(* Logix 5000 project; controller Nut_Filling_Station Emulate 5570 rev 33.11; software revision 33.03 *)

TASK MainTask (continuous, watchdog 500 ms) : MainProgram

MODULES
   Local : Emulate 5570 (ICP 3, rev 33.11)
END_MODULES

VAR_GLOBAL   (* controller tags *)
   Conveyor_Run : BOOL;   // Conveyor motor command
   Entry_PE : BOOL;   // Box at label-reading position
   Exit_PE : BOOL;   // Box at exit
   Green_Label : BOOL;   // Green label detected
   Peanut_Box_Count : COUNTER := (PRE := 1000);   // Counts completed peanut boxes
   Peanut_Filled_Up : BOOL;   // Peanut station reports target weight reached
   Peanut_Open : BOOL;   // Peanut hopper valve command
   Peanut_PE : BOOL;   // Box underneath peanut hopper
   Peanut_Total_kg : REAL;   // Total peanut kilograms packed
   Red_Label : BOOL;   // Red label detected
   Reset_Counts_PB : BOOL;   // Clears production counts
   Reset_PB : BOOL;   // Reset sequence
   Run_Enable : BOOL;   // Automatic operation enabled
   Start_PB : BOOL;   // Start pushbutton
   Step : DINT;   // Current sequence step
   Step_Scan : DINT;   // Step captured at start of this scan
   Stop_OK : BOOL;   // 1 when Stop is released
   Walnut_Box_Count : COUNTER := (PRE := 1000);   // Counts completed walnut boxes
   Walnut_Filled_Up : BOOL;   // Walnut station reports target weight reached
   Walnut_Open : BOOL;   // Walnut hopper valve command
   Walnut_PE : BOOL;   // Box underneath walnut hopper
   Walnut_Total_kg : REAL;   // Total walnut kilograms packed
END_VAR

PROGRAM MainProgram   (* main routine MainRoutine *)

ROUTINE MainRoutine   (* ladder *)
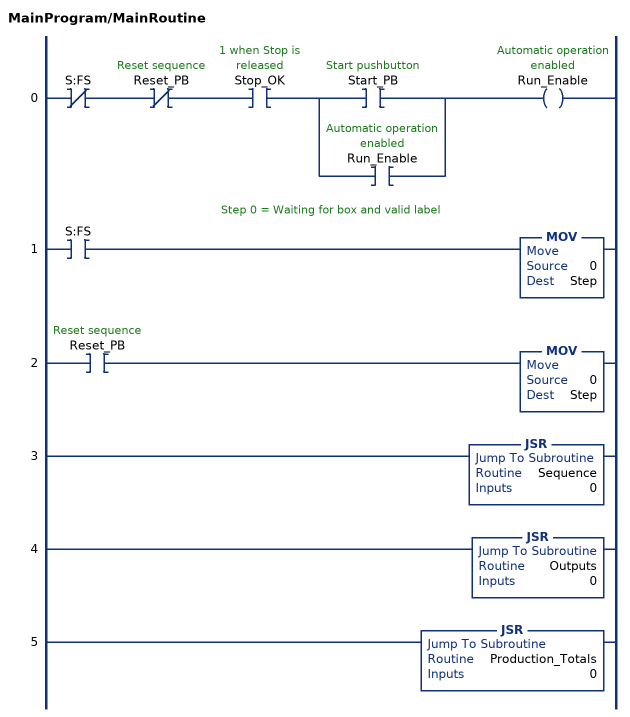
   0: XIO(S:FS)XIO(Reset_PB)XIC(Stop_OK)[XIC(Start_PB) ,XIC(Run_Enable) ]OTE(Run_Enable);
   // Step 0 = Waiting for box and valid label
   1: XIC(S:FS)MOV(0,Step);
   2: XIC(Reset_PB)MOV(0,Step);
   3: JSR(Sequence,0);
   4: JSR(Outputs,0);
   5: JSR(Production_Totals,0);
END_ROUTINE

ROUTINE Outputs   (* ladder *)
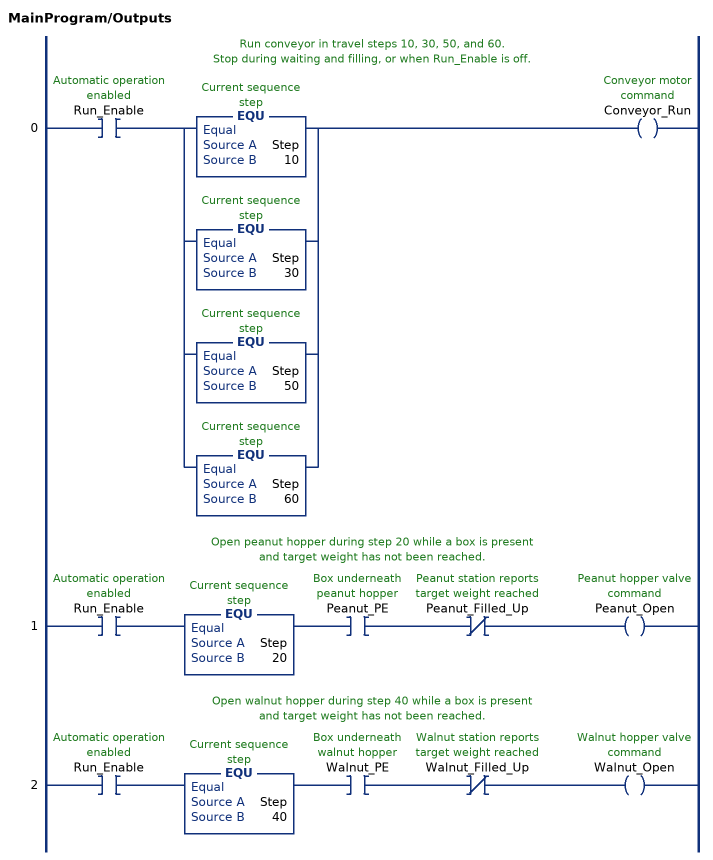
   // Run conveyor in travel steps 10, 30, 50, and 60.
   // Stop during waiting and filling, or when Run_Enable is off.
   0: XIC(Run_Enable)[EQU(Step,10) ,EQU(Step,30) ,EQU(Step,50) ,EQU(Step,60) ]OTE(Conveyor_Run);
   // Open peanut hopper during step 20 while a box is present
   // and target weight has not been reached.
   1: XIC(Run_Enable)EQU(Step,20)XIC(Peanut_PE)XIO(Peanut_Filled_Up)OTE(Peanut_Open);
   // Open walnut hopper during step 40 while a box is present
   //  and target weight has not been reached.
   2: XIC(Run_Enable)EQU(Step,40)XIC(Walnut_PE)XIO(Walnut_Filled_Up)OTE(Walnut_Open);
END_ROUTINE

ROUTINE Production_Totals   (* ladder *)
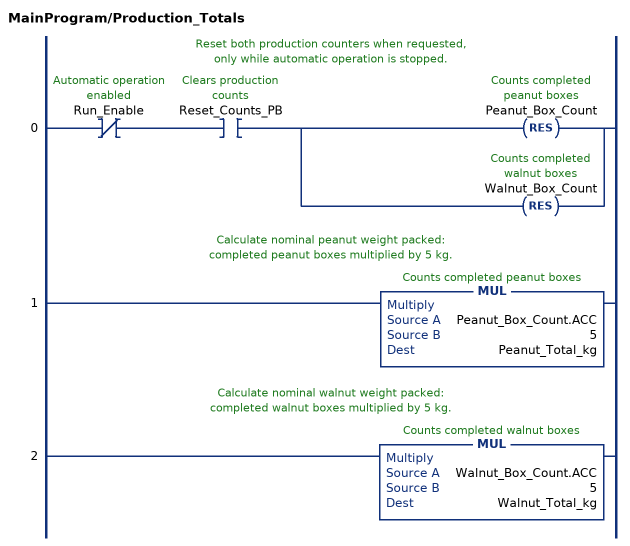
   // Reset both production counters when requested,
   // only while automatic operation is stopped.
   0: XIO(Run_Enable)XIC(Reset_Counts_PB)[RES(Peanut_Box_Count) ,RES(Walnut_Box_Count) ];
   // Calculate nominal peanut weight packed:
   // completed peanut boxes multiplied by 5 kg.
   1: MUL(Peanut_Box_Count.ACC,5,Peanut_Total_kg);
   // Calculate nominal walnut weight packed:
   // completed walnut boxes multiplied by 5 kg.
   2: MUL(Walnut_Box_Count.ACC,5,Walnut_Total_kg);
END_ROUTINE

ROUTINE Sequence   (* ladder *)
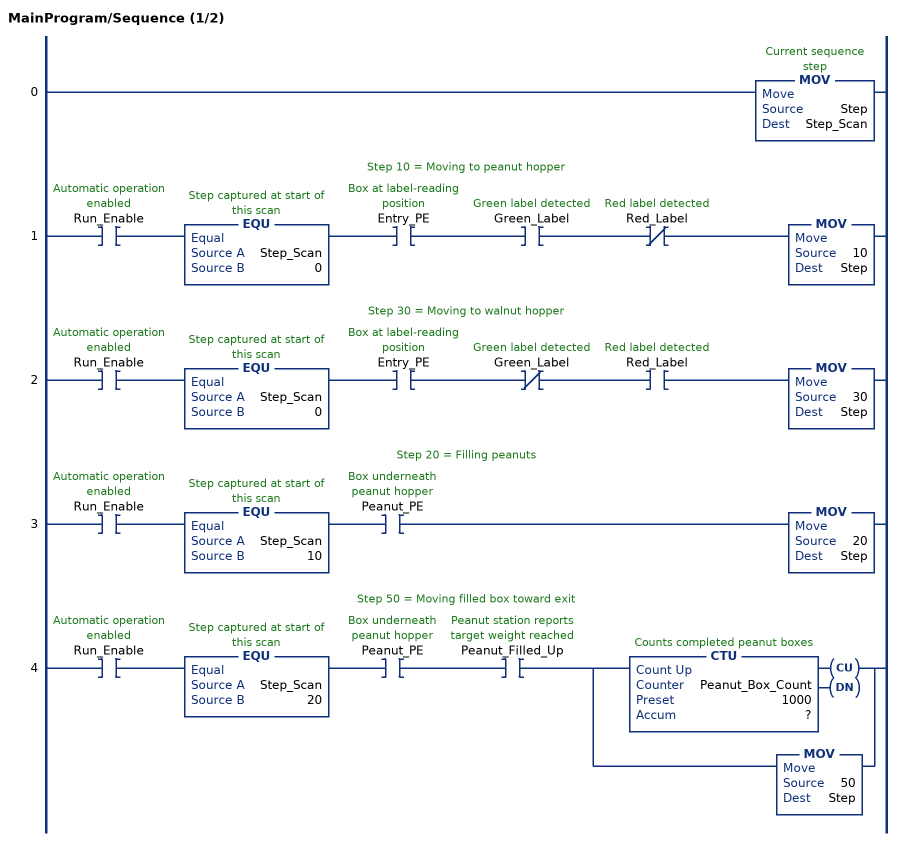
   0: MOV(Step,Step_Scan);
   // Step 10 = Moving to peanut hopper
   1: XIC(Run_Enable)EQU(Step_Scan,0)XIC(Entry_PE)XIC(Green_Label)XIO(Red_Label)MOV(10,Step);
   // Step 30 = Moving to walnut hopper
   2: XIC(Run_Enable)EQU(Step_Scan,0)XIC(Entry_PE)XIO(Green_Label)XIC(Red_Label)MOV(30,Step);
   // Step 20 = Filling peanuts
   3: XIC(Run_Enable)EQU(Step_Scan,10)XIC(Peanut_PE)MOV(20,Step);
   // Step 50 = Moving filled box toward exit
   4: XIC(Run_Enable)EQU(Step_Scan,20)XIC(Peanut_PE)XIC(Peanut_Filled_Up)[CTU(Peanut_Box_Count,?,?) ,MOV(50,Step) ];
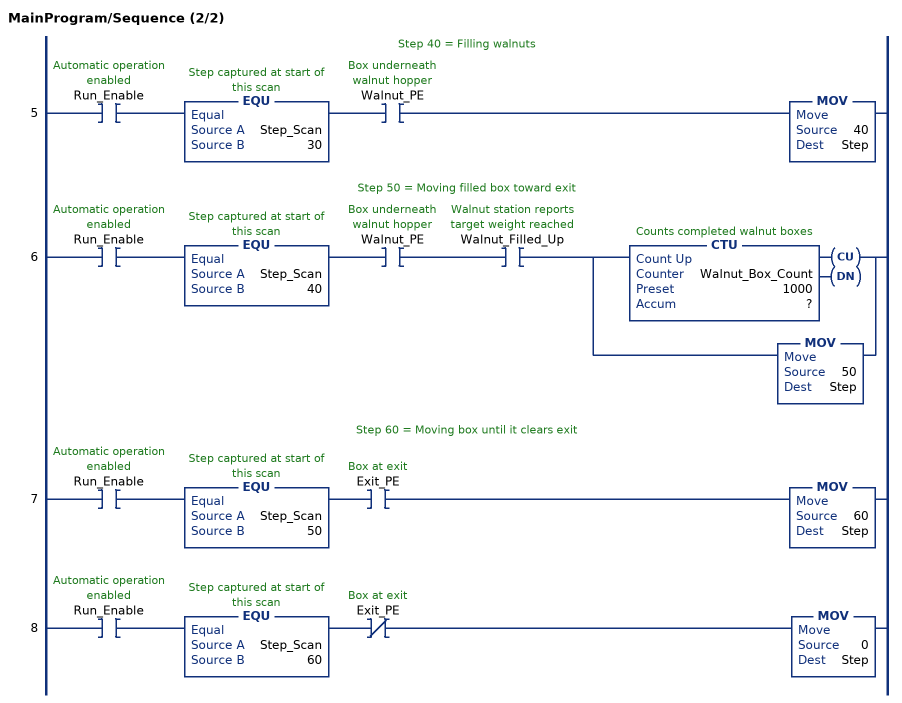
   // Step 40 = Filling walnuts
   5: XIC(Run_Enable)EQU(Step_Scan,30)XIC(Walnut_PE)MOV(40,Step);
   // Step 50 = Moving filled box toward exit
   6: XIC(Run_Enable)EQU(Step_Scan,40)XIC(Walnut_PE)XIC(Walnut_Filled_Up)[CTU(Walnut_Box_Count,?,?) ,MOV(50,Step) ];
   // Step 60 = Moving box until it clears exit
   7: XIC(Run_Enable)EQU(Step_Scan,50)XIC(Exit_PE)MOV(60,Step);
   8: XIC(Run_Enable)EQU(Step_Scan,60)XIO(Exit_PE)MOV(0,Step);
END_ROUTINE
END_PROGRAM
